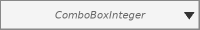
VISUALIZATION VISU_HELPER_Combobox_eSignalform  // 200x30
VAR_IN_OUT
    varEnum : eReglertyp;
END_VAR
    ComboBoxInteger (0,0 200x30), variable: varEnum, text list: 'TextListForCombobox_eSignalform'
END_VISUALIZATION

(* stored: Version 1.1.0.1, ProductVersion 3.1.4024.12
   Visu VISU_HELPER_Combobox_eSignalform: Id {9f55e8ba-d176-4ceb-af27-fcdef4f9c227} *)
